// TIA Portal V21 export
DATA_BLOCK "PV"   // DB194
{ S7_Optimized_Access := 'TRUE' }
// stored: MemoryReserve 100
   VAR
      "CHAMBER PRESS" : Real;
      "DRAIN TEMP" : Real;
      "JACKET TEMP" : Real;
      VACCUM : Real;
      "CHAMBER TEMP1" : Real;
      "CHAMBER TEMP2" : Real;
      "CHAMBER TEMP3" : Real;
      "CHAMBER TEMP4" : Real;
      "DOOR1 PRESS" : Real;
      "DOOR2 PRESS" : Real;
      "JACKET PRESS" : Real;
      "DOOR1 VACCUM" : Real;
      "DOOR2 VACCUM" : Real;
      "JACKET VACCUM" : Real;
   END_VAR
BEGIN
END_DATA_BLOCK
